TYPE ST_MotorSSErrors :
STRUCT	
	SofstarterFailure		: BOOL;
	Maintenance				: BOOL;
END_STRUCT
END_TYPE

(* stored: Version 1.1.0.1, ProductVersion 3.1.4020.12
   DUT ST_MotorSSErrors: Id {7c0a491f-2efe-4ca3-8bc2-dee14206f7db} *)
